// Mitsubishi GX Works2 project: 241206   PLC: Q02U

PROGRAM MAIN
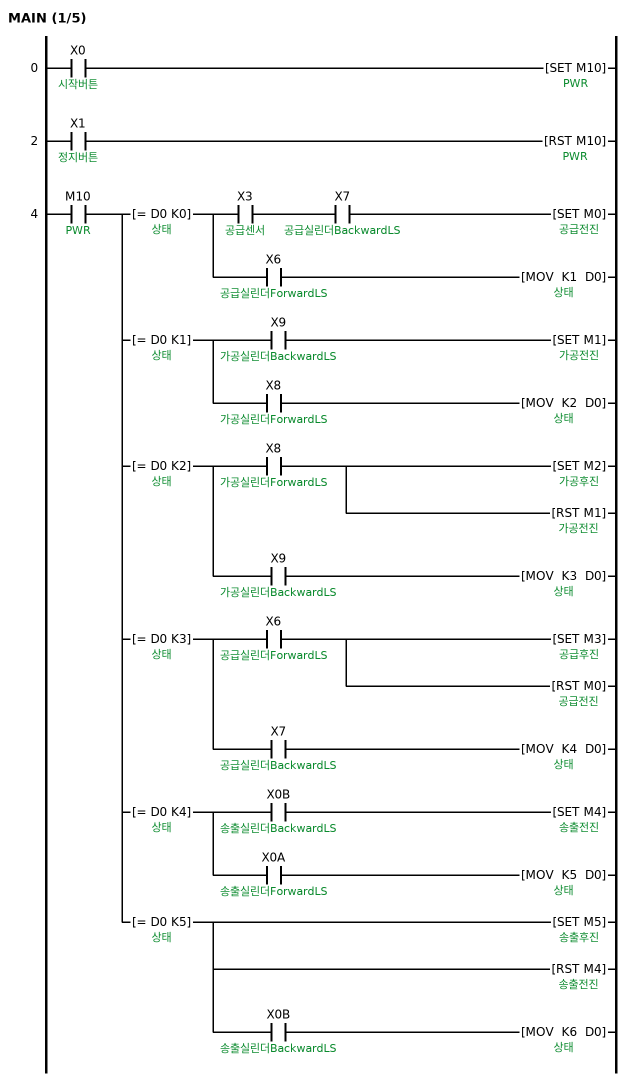
0     LD      X0  ; 시작버튼
      SET     M10  ; PWR
2     LD      X1  ; 정지버튼
      RST     M10  ; PWR
4     LD      M10  ; PWR
      MPS
      AND=    D0 K0  ; 상태
      MPS
      AND     X3  ; 공급센서
      AND     X7  ; 공급실린더BackwardLS
      SET     M0  ; 공급전진
      MPP
      AND     X6  ; 공급실린더ForwardLS
      MOV     K1 D0
      MRD
      AND=    D0 K1  ; 상태
      MPS
      AND     X9  ; 가공실린더BackwardLS
      SET     M1  ; 가공전진
      MPP
      AND     X8  ; 가공실린더ForwardLS
      MOV     K2 D0
      MRD
      AND=    D0 K2  ; 상태
      MPS
      AND     X8  ; 가공실린더ForwardLS
      SET     M2  ; 가공후진
      RST     M1  ; 가공전진
      MPP
      AND     X9  ; 가공실린더BackwardLS
      MOV     K3 D0
      MRD
      AND=    D0 K3  ; 상태
      MPS
      AND     X6  ; 공급실린더ForwardLS
      SET     M3  ; 공급후진
      RST     M0  ; 공급전진
      MPP
      AND     X7  ; 공급실린더BackwardLS
      MOV     K4 D0
      MRD
      AND=    D0 K4  ; 상태
      MPS
      AND     X0B  ; 송출실린더BackwardLS
      SET     M4  ; 송출전진
      MPP
      AND     X0A  ; 송출실린더ForwardLS
      MOV     K5 D0
      MPP
      AND=    D0 K5  ; 상태
      SET     M5  ; 송출후진
      RST     M4  ; 송출전진
      AND     X0B  ; 송출실린더BackwardLS
      MOV     K6 D0
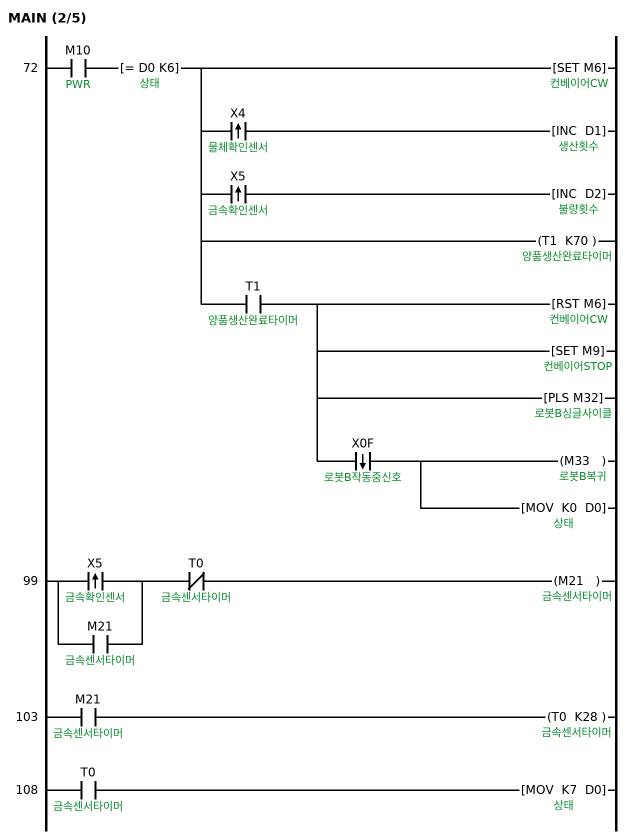
72    LD      M10  ; PWR
      AND=    D0 K6  ; 상태
      SET     M6  ; 컨베이어CW
      MPS
      ANDP    X4  ; 물체확인센서
      INC     D1  ; 생산횟수
      MRD
      ANDP    X5  ; 금속확인센서
      INC     D2  ; 불량횟수
      MPP
      OUT     T1 K70  ; 양품생산완료타이머
      AND     T1  ; 양품생산완료타이머
      RST     M6  ; 컨베이어CW
      SET     M9  ; 컨베이어STOP
      PLS     M32  ; 로봇B싱글사이클
      ANDF    X0F  ; 로봇B작동중신호
      OUT     M33  ; 로봇B복귀
      MOV     K0 D0
99    LDP     X5  ; 금속확인센서
      OR      M21  ; 금속센서타이머
      ANI     T0  ; 금속센서타이머
      OUT     M21  ; 금속센서타이머
103   LD      M21  ; 금속센서타이머
      OUT     T0 K28  ; 금속센서타이머
108   LD      T0  ; 금속센서타이머
      MOV     K7 D0
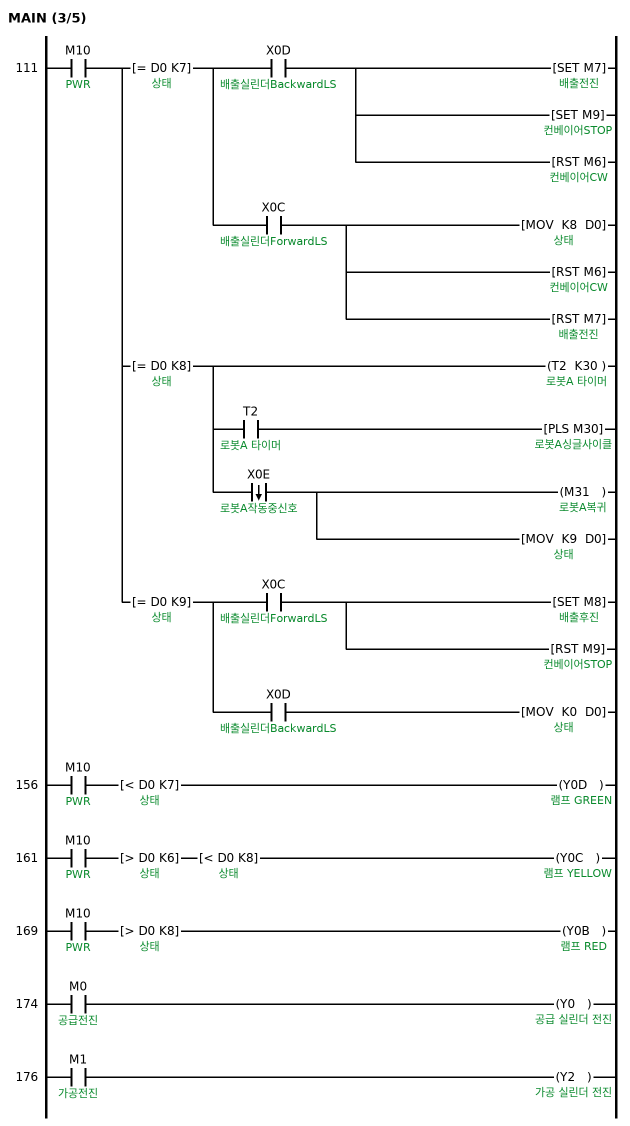
111   LD      M10  ; PWR
      MPS
      AND=    D0 K7  ; 상태
      MPS
      AND     X0D  ; 배출실린더BackwardLS
      SET     M7  ; 배출전진
      SET     M9  ; 컨베이어STOP
      RST     M6  ; 컨베이어CW
      MPP
      AND     X0C  ; 배출실린더ForwardLS
      MOV     K8 D0
      RST     M6  ; 컨베이어CW
      RST     M7  ; 배출전진
      MRD
      AND=    D0 K8  ; 상태
      OUT     T2 K30  ; 로봇A 타이머
      MPS
      AND     T2  ; 로봇A 타이머
      PLS     M30  ; 로봇A싱글사이클
      MPP
      ANDF    X0E  ; 로봇A작동중신호
      OUT     M31  ; 로봇A복귀
      MOV     K9 D0
      MPP
      AND=    D0 K9  ; 상태
      MPS
      AND     X0C  ; 배출실린더ForwardLS
      SET     M8  ; 배출후진
      RST     M9  ; 컨베이어STOP
      MPP
      AND     X0D  ; 배출실린더BackwardLS
      MOV     K0 D0
156   LD      M10  ; PWR
      AND<    D0 K7  ; 상태
      OUT     Y0D  ; 램프 GREEN
161   LD      M10  ; PWR
      AND>    D0 K6  ; 상태
      AND<    D0 K8  ; 상태
      OUT     Y0C  ; 램프 YELLOW
169   LD      M10  ; PWR
      AND>    D0 K8  ; 상태
      OUT     Y0B  ; 램프 RED
174   LD      M0  ; 공급전진
      OUT     Y0  ; 공급 실린더 전진
176   LD      M1  ; 가공전진
      OUT     Y2  ; 가공 실린더 전진
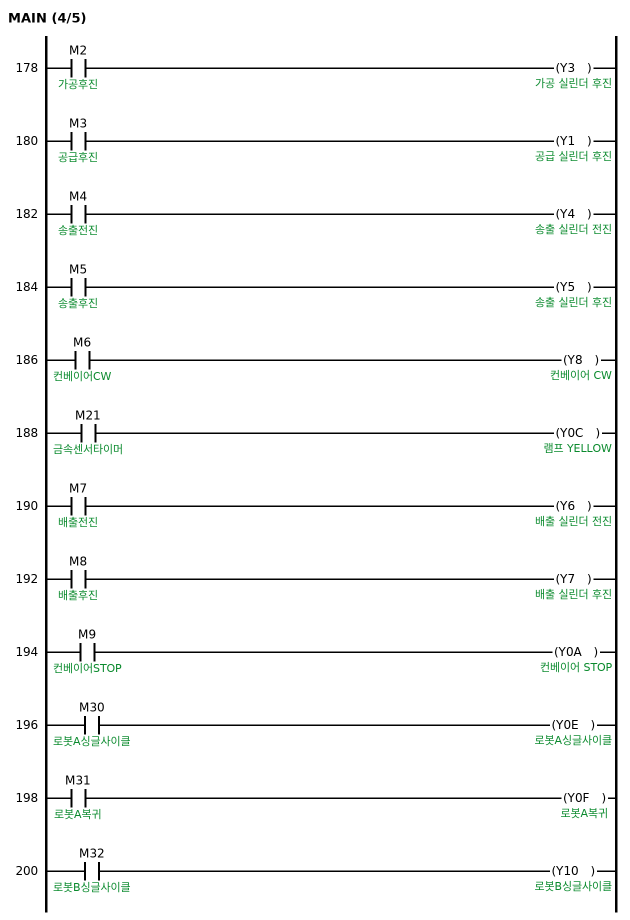
178   LD      M2  ; 가공후진
      OUT     Y3  ; 가공 실린더 후진
180   LD      M3  ; 공급후진
      OUT     Y1  ; 공급 실린더 후진
182   LD      M4  ; 송출전진
      OUT     Y4  ; 송출 실린더 전진
184   LD      M5  ; 송출후진
      OUT     Y5  ; 송출 실린더 후진
186   LD      M6  ; 컨베이어CW
      OUT     Y8  ; 컨베이어 CW
188   LD      M21  ; 금속센서타이머
      OUT     Y0C  ; 램프 YELLOW
190   LD      M7  ; 배출전진
      OUT     Y6  ; 배출 실린더 전진
192   LD      M8  ; 배출후진
      OUT     Y7  ; 배출 실린더 후진
194   LD      M9  ; 컨베이어STOP
      OUT     Y0A  ; 컨베이어 STOP
196   LD      M30  ; 로봇A싱글사이클
      OUT     Y0E  ; 로봇A싱글사이클
198   LD      M31  ; 로봇A복귀
      OUT     Y0F  ; 로봇A복귀
200   LD      M32  ; 로봇B싱글사이클
      OUT     Y10  ; 로봇B싱글사이클
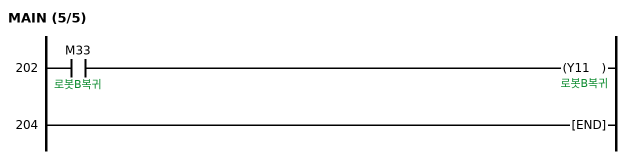
202   LD      M33  ; 로봇B복귀
      OUT     Y11  ; 로봇B복귀
204   END
END_PROGRAM

// device comments not shown above
X2  ; 긴급정지버튼
Y9  ; 컨베이어 CCW
M20  ; 컨베이어 CW
M22  ; 컨베이어 STOP
